TYPE ST_SP_RecordReturn :
STRUCT
	tableId: UDINT;
	//classId: STRING(3);
	errorId: STRING(3);
	severity: BYTE;
	errorMsgShort: T_MaxString;
	errorMsgLong: T_MaxString;
	remediationMsg: T_MaxString;
	telegramSending: STRING(1);
	hmiErrorShow: STRING(1);
END_STRUCT
END_TYPE

(* stored: Version 1.1.0.1, ProductVersion 3.1.4024.12
   DUT ST_SP_RecordReturn: Id {bfb6bbb1-2cda-45da-b052-79bbf3658d1e} *)
